INTERFACE ITF_BaseTopElement EXTENDS ITF_BaseGroupElement, ITF_BaseSaMStateMethod

METHOD PUBLIC LinkSaM : BOOL
VAR_INPUT
	fbSAM				: ITF_BaseSAM;
END_VAR
END_METHOD

END_INTERFACE

(* stored: Version 1.1.0.1
   Itf ITF_BaseTopElement: Id {2822f205-b986-005f-04be-ccc64a012929}
   Method LinkSaM: Id {afe7878d-4995-0f53-2961-aff4e9d5c093} *)
